TYPE DUT_TASK :
STRUCT
	///Name of the Task
	Name: STRING(80);
	///Free to use = TRUE, busy to use =FALSE
	Dummy: BOOL := TRUE;
	///Identification number of the Task
	TaskID: INT;
	///Identification number of the Recipe
	RecipeID: INT;
	///Range of Skill in the TASK
	Skill: ARRAY[0..TaskSkillCnt] OF DUT_SKILL;
	///When occurs the action
	Timestamp: STRING(80);
	///State of the TASK e.g (unassigned, assigned, waitingForSkillReady, inProgress, done, aborted, error)
	State: DUT_TASKSTATE := 0;
END_STRUCT
END_TYPE

(* stored: Version 1.1.0.1, ProductVersion 3.1.0.25
   DUT DUT_TASK: Id {8a9ce35f-8ebe-4dbb-b09a-05b0b2286129} *)
